// TIA Portal V17 export
FUNCTION "FC_烧嘴报警" : Void   // FC, LAD
{ S7_Optimized_Access := 'TRUE' }
   VAR_TEMP   // added for the SCL form of the ladder/FBD networks
      _w1 : Bool;
      _w2 : Bool;
   END_VAR
BEGIN

REGION Network 1: 故障反馈汇总与蜂鸣器报警
   // 任意烧嘴故障反馈上升沿时置位蜂鸣器输出
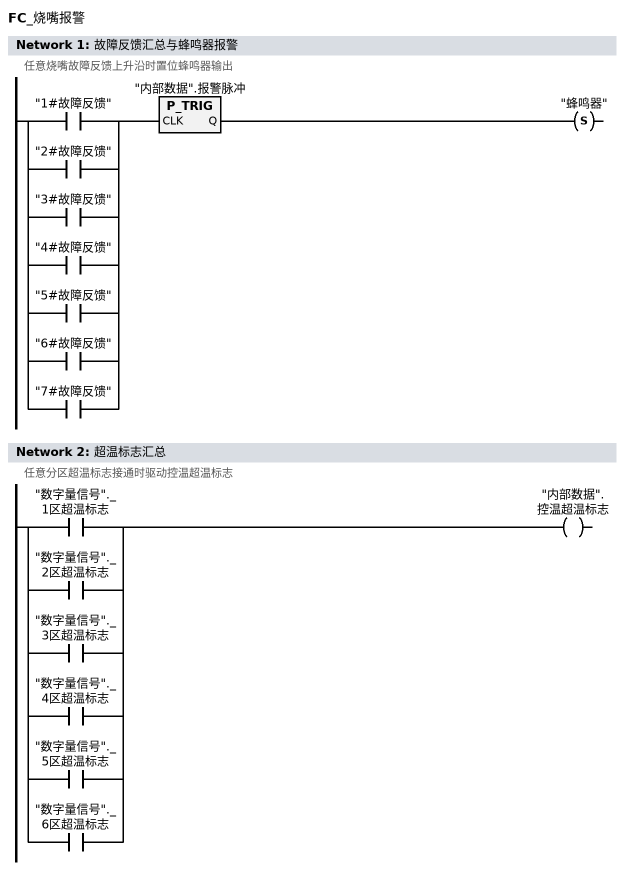
   RUNG wire#powerrail
      Contact( "1#故障反馈" )
      wire#w1
      P_Trig( "内部数据".报警脉冲 )
      S_Coil( "蜂鸣器" )
   END_RUNG
   RUNG wire#powerrail
      Contact( "2#故障反馈" )
   END_RUNG wire#w1
   RUNG wire#powerrail
      Contact( "3#故障反馈" )
   END_RUNG wire#w1
   RUNG wire#powerrail
      Contact( "4#故障反馈" )
   END_RUNG wire#w1
   RUNG wire#powerrail
      Contact( "5#故障反馈" )
   END_RUNG wire#w1
   RUNG wire#powerrail
      Contact( "6#故障反馈" )
   END_RUNG wire#w1
   RUNG wire#powerrail
      Contact( "7#故障反馈" )
   END_RUNG wire#w1
   // the same network as SCL:
   #_w1 := "1#故障反馈" OR "2#故障反馈" OR "3#故障反馈" OR "4#故障反馈" OR "5#故障反馈" OR "6#故障反馈" OR "7#故障反馈";
   #_w2 := #_w1 AND NOT "内部数据".报警脉冲;   // rising edge
   "内部数据".报警脉冲 := #_w1;
   IF #_w2 THEN "蜂鸣器" := TRUE; END_IF;
END_REGION

REGION Network 2: 超温标志汇总
   // 任意分区超温标志接通时驱动控温超温标志
   RUNG wire#powerrail
      Contact( "数字量信号"._1区超温标志 )
      wire#w1
      Coil( "内部数据".控温超温标志 )
   END_RUNG
   RUNG wire#powerrail
      Contact( "数字量信号"._2区超温标志 )
   END_RUNG wire#w1
   RUNG wire#powerrail
      Contact( "数字量信号"._3区超温标志 )
   END_RUNG wire#w1
   RUNG wire#powerrail
      Contact( "数字量信号"._4区超温标志 )
   END_RUNG wire#w1
   RUNG wire#powerrail
      Contact( "数字量信号"._5区超温标志 )
   END_RUNG wire#w1
   RUNG wire#powerrail
      Contact( "数字量信号"._6区超温标志 )
   END_RUNG wire#w1
   // the same network as SCL:
   "内部数据".控温超温标志 := "数字量信号"._1区超温标志 OR "数字量信号"._2区超温标志 OR "数字量信号"._3区超温标志 OR "数字量信号"._4区超温标志 OR "数字量信号"._5区超温标志 OR "数字量信号"._6区超温标志;
END_REGION
END_FUNCTION
